PROGRAM PRG_3_LOG
VAR
      fbLogHandler: FB_LogHandler;
END_VAR


fbLogHandler();

END_PROGRAM

(* stored: Version 1.1.0.1
   POU PRG_3_LOG: Id {48e166b6-5fab-41f0-8dbc-ebe24636762e}, SpecialFunc None *)
